INTERFACE I_Cyclic EXTENDS I_Base

METHOD CyclicLogic : BOOL
VAR_INPUT
END_VAR
END_METHOD

PROPERTY InitCompleted : Bool
GET
END_GET
END_PROPERTY

END_INTERFACE

(* stored: Version 1.1.0.1, ProductVersion 3.1.4024.14
   Itf I_Cyclic: Id {98a1eaf4-08c0-471e-82d4-eb2d7fb645b7}
   Folder Methods: Id {ae7d0a2c-a37f-41e8-bbad-27f20ac153fe}
   Folder Properties: Id {2134fa10-45da-4a16-9ef1-542792a88b42}
   Method CyclicLogic: Id {ab56a435-5d01-41e9-afff-00b72d8e3c0f}
   Property InitCompleted: Id {754992be-0c43-4d96-b5c5-0dc5aa945203}
   Get Get: Id {164716b1-2930-4265-8b52-d8dd9f3d8dc3} *)
